PROGRAM LinkHWIO
VAR
	
END_VAR

GVL_SignalHanlding.fbHandleStartBtn.bSignalInput := GVL_Machine.HWIO.HWInput.StartBtn OR GVL_SignalHanlding.fbHandleStartBtn.bSignalInput;
GVL_SignalHanlding.fbHandleStartBtn.SignalEnable(bSignalLocalEnable := (GVL_Machine.machineMode = MachineMode.Auto));
GVL_SignalHanlding.fbHandleStartBtn.SetOutput();


//==========Hardware signal inPauseBtn handle==========
(*GVL_SignalHanlding.inPauseBtnHandling.bSignalInput := ((GVL_Machine.HWIO.HWInput.PauseBtn OR GVL_SignalHanlding.fbPauseUI.bSignalOutput
														 OR GVL_SignalHanlding.inPauseBtnHandling.bSignalInput) AND NOT (GVL_Machine.HWIO.HWInput.StartBtn));
														 
GVL_SignalHanlding.inPauseBtnHandling.SignalEnable(bSignalLocalEnable := (GVL_Machine.machineMode = MachineMode.Auto OR GVL_Machine.machineMode = MachineMode.Manual));
GVL_SignalHanlding.inPauseBtnHandling.SetOutput();  *)

GVL_SignalHanlding.inPauseBtnHandling.bSignalInput := GVL_Machine.HWIO.HWInput.PauseBtn  OR GVL_SignalHanlding.inPauseBtnHandling.bSignalOutput;
GVL_SignalHanlding.inPauseBtnHandling.SignalEnable(bSignalLocalEnable :=(GVL_Machine.machineMode = MachineMode.Auto) AND NOT GVL_Machine.HWIO.HWInput.StartBtn);
GVL_SignalHanlding.inPauseBtnHandling.SetOutput(); 
//==========Hardware signal inPause handle==========


//==========Hardware signal inStop handle==========
GVL_SignalHanlding.inStopBtnHandling.bSignalInput := GVL_Machine.HWIO.HWInput.StopBtn OR GVL_SignalHanlding.inStopBtnHandling.bSignalOutput;
GVL_SignalHanlding.inStopBtnHandling.SignalEnable(bSignalLocalEnable := (GVL_Machine.machineMode = MachineMode.Auto) AND NOT GVL_Machine.HWIO.HWInput.StartBtn);
GVL_SignalHanlding.inStopBtnHandling.SetOutput();
//==========Hardware signal inStop handle==========

END_PROGRAM

(* stored: Version 1.1.0.1, ProductVersion 3.1.4022.16
   POU LinkHWIO: Id {ca7c5f8c-3572-4336-a709-121a682bf16f}, SpecialFunc None *)
